Fanuc KAREL source: kt00303.compact.KL

PROGRAM KT00303
%STACKSIZE=65535
%PRIORITY=65535
%NOLOCKGROUP
VAR
Y1 : ARRAY[2] OF BYTE
I2 : INTEGER
OUT : BOOLEAN
BEGIN
Y1[1]=2
I2=3
OUT=(Y1[1] <> I2)
END KT00303
